{attribute addProperty BoxType "IODEVICETYPE_ETHERCATPROT"}
{attribute addProperty Id "Beckhoff_EL1xxxBeckhoff_EL1xxx_78602F53606967587Beckhoff_EL2xxxBeckhoff_EL2xxx_69484E48239162989.5Beckhoff_EL3xxxBeckhoff_EL3xxx_8EB68CB4123221540.25Beckhoff_EL3xxx_0030Beckhoff_EL3xxx_0030_C3F11E951587198.375Beckhoff_EL4xxxBeckhoff_EL4xxx_1F5CAB3C192402405Beckhoff_EL5xxxBeckhoff_EL5xxx_6457D9C7191042388Beckhoff_EL6xxxBeckhoff_EL6xxx_DCB17FC9205932574.125Beckhoff_EL7xxxBeckhoff_EL7xxx_252AF501129881623.5Beckhoff_EL9xxxBeckhoff_EL9xxx_69A9CD637432929Beckhoff_EL15xxBeckhoff_EL15xx_D9B38BDD3752469Beckhoff_EL19xxBeckhoff_EL19xx_71C3041123229Beckhoff_EL25xxBeckhoff_EL25xx_79BFBDD6175522194Beckhoff_EL29xxBeckhoff_EL29xx_49DA042452065Beckhoff_EL30xxBeckhoff_EL30xx_41983985360474505.875Beckhoff_EL31xxBeckhoff_EL31xx_18A76DD1202642533Beckhoff_EL32xxBeckhoff_EL32xx_1D50FE80173142164.25Beckhoff_EL33xxBeckhoff_EL33xx_5EBAF070191522394Beckhoff_EL34xxBeckhoff_EL34xx_71FD10A09253611567Beckhoff_EL37xxBeckhoff_EL37xx_EF75DD5D159601995Beckhoff_EL47xxBeckhoff_EL47xx_AD32B54A2352294Beckhoff_EL66xxBeckhoff_EL66xx_BDCA255982721034Beckhoff_EL67xxBeckhoff_EL67xx_7CBCD6777728966Beckhoff_EL68xxBeckhoff_EL68xx_60CF9DE5286163577Beckhoff_EL69xxBeckhoff_EL69xx_FB8F557D1584198Beckhoff_EL72xxBeckhoff_EL72xx_6413AB37270643383Beckhoff_EL73xxBeckhoff_EL73xx_43145A975728716Beckhoff_EL99xxBeckhoff_EL99xx_AE62663A8010SyncUnitsSyncUnits_641B4EFA149041863InputsInputs_C75D3FEC1280160OutputsOutputs_47D1E803848106InfoDataInfoData_45F98C5022428"}
{attribute addProperty CRC "1065899834"}
{attribute addProperty SizeInBites "499887"}
{attribute addProperty SizeInBytes "62485.875"}
TYPE EtherCAT_Master_ELxxxx_3F88573A :
STRUCT
	{attribute addProperty Name "Beckhoff_EL1xxx"}
	Beckhoff_EL1xxx : Beckhoff_EL1xxx_78602F53;
	{attribute addProperty Name "Beckhoff_EL2xxx"}
	Beckhoff_EL2xxx : Beckhoff_EL2xxx_69484E48;
	{attribute addProperty Name "Beckhoff_EL3xxx"}
	Beckhoff_EL3xxx : Beckhoff_EL3xxx_8EB68CB4;
	{attribute addProperty Name "Beckhoff_EL3xxx_0030"}
	Beckhoff_EL3xxx_0030 : Beckhoff_EL3xxx_0030_C3F11E95;
	{attribute addProperty Name "Beckhoff_EL4xxx"}
	Beckhoff_EL4xxx : Beckhoff_EL4xxx_1F5CAB3C;
	{attribute addProperty Name "Beckhoff_EL5xxx"}
	Beckhoff_EL5xxx : Beckhoff_EL5xxx_6457D9C7;
	{attribute addProperty Name "Beckhoff_EL6xxx"}
	Beckhoff_EL6xxx : Beckhoff_EL6xxx_DCB17FC9;
	{attribute addProperty Name "Beckhoff_EL7xxx"}
	Beckhoff_EL7xxx : Beckhoff_EL7xxx_252AF501;
	{attribute addProperty Name "Beckhoff_EL9xxx"}
	Beckhoff_EL9xxx : Beckhoff_EL9xxx_69A9CD63;
	{attribute addProperty Name "Beckhoff_EL15xx"}
	Beckhoff_EL15xx : Beckhoff_EL15xx_D9B38BDD;
	{attribute addProperty Name "Beckhoff_EL19xx"}
	Beckhoff_EL19xx : Beckhoff_EL19xx_71C30411;
	{attribute addProperty Name "Beckhoff_EL25xx"}
	Beckhoff_EL25xx : Beckhoff_EL25xx_79BFBDD6;
	{attribute addProperty Name "Beckhoff_EL29xx"}
	Beckhoff_EL29xx : Beckhoff_EL29xx_49DA0424;
	{attribute addProperty Name "Beckhoff_EL30xx"}
	Beckhoff_EL30xx : Beckhoff_EL30xx_41983985;
	{attribute addProperty Name "Beckhoff_EL31xx"}
	Beckhoff_EL31xx : Beckhoff_EL31xx_18A76DD1;
	{attribute addProperty Name "Beckhoff_EL32xx"}
	Beckhoff_EL32xx : Beckhoff_EL32xx_1D50FE80;
	{attribute addProperty Name "Beckhoff_EL33xx"}
	Beckhoff_EL33xx : Beckhoff_EL33xx_5EBAF070;
	{attribute addProperty Name "Beckhoff_EL34xx"}
	Beckhoff_EL34xx : Beckhoff_EL34xx_71FD10A0;
	{attribute addProperty Name "Beckhoff_EL37xx"}
	Beckhoff_EL37xx : Beckhoff_EL37xx_EF75DD5D;
	{attribute addProperty Name "Beckhoff_EL47xx"}
	Beckhoff_EL47xx : Beckhoff_EL47xx_AD32B54A;
	{attribute addProperty Name "Beckhoff_EL66xx"}
	Beckhoff_EL66xx : Beckhoff_EL66xx_BDCA2559;
	{attribute addProperty Name "Beckhoff_EL67xx"}
	Beckhoff_EL67xx : Beckhoff_EL67xx_7CBCD677;
	{attribute addProperty Name "Beckhoff_EL68xx"}
	Beckhoff_EL68xx : Beckhoff_EL68xx_60CF9DE5;
	{attribute addProperty Name "Beckhoff_EL69xx"}
	Beckhoff_EL69xx : Beckhoff_EL69xx_FB8F557D;
	{attribute addProperty Name "Beckhoff_EL72xx"}
	Beckhoff_EL72xx : Beckhoff_EL72xx_6413AB37;
	{attribute addProperty Name "Beckhoff_EL73xx"}
	Beckhoff_EL73xx : Beckhoff_EL73xx_43145A97;
	{attribute addProperty Name "Beckhoff_EL99xx"}
	Beckhoff_EL99xx : Beckhoff_EL99xx_AE62663A;
	{attribute addProperty Name "SyncUnits"}
	SyncUnits : SyncUnits_641B4EFA;
	{attribute addProperty Name "Inputs"}
	Inputs : Inputs_C75D3FEC;
	{attribute addProperty Name "Outputs"}
	Outputs : Outputs_47D1E803;
	{attribute addProperty Name "InfoData"}
	InfoData : InfoData_45F98C50;
END_STRUCT
END_TYPE

(* stored: Version 1.2.0.0, ProductVersion 3.1.4024.9
   DUT EtherCAT_Master_ELxxxx_3F88573A: Id {ee7294b2-38de-4303-ab58-261f1d2ccafc} *)
